(* PLC project First Steps, Beremiz Beremiz 1 *)
(* stored: creationDateTime 2016-10-24T18:09:22, modificationDateTime 2024-12-18T14:47:09 *)

PROGRAM plc_prg
  VAR
    LocalVar0 : DINT := 0;
  END_VAR
  VAR
    LocalVar1 AT %QD0.2 : DINT;
    LocalVar2 AT %ID0.2 : DINT;
  END_VAR
  VAR
    python_eval0 : python_eval;
    python_eval1 : python_eval;
  END_VAR
  VAR  (* added by the conversion: wires and edge detectors of the diagram *)
    _GT8_OUT : BOOL;
  END_VAR

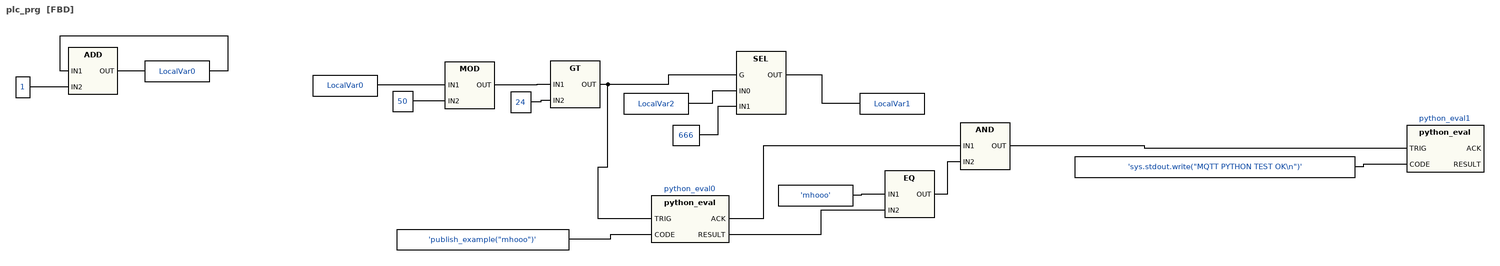
(* FBD diagram, written out as Structured Text *)
LocalVar0 := LocalVar0 + 1;
_GT8_OUT := LocalVar0 MOD 50 > 24;
LocalVar1 := SEL(_GT8_OUT, LocalVar2, 666);
python_eval0(TRIG := _GT8_OUT, CODE := 'publish_example("mhooo")');
python_eval1(TRIG := python_eval0.ACK AND 'mhooo' = python_eval0.RESULT, CODE := 'sys.stdout.write("MQTT PYTHON TEST OK\n")');
END_PROGRAM

CONFIGURATION config
  VAR_GLOBAL CONSTANT
    ResetCounterValue : INT := 17;
  END_VAR
  RESOURCE resource1 ON PLC
    TASK plc_task(INTERVAL := T#100ms, PRIORITY := 1);
    PROGRAM plc_task_instance WITH plc_task : plc_prg;
  END_RESOURCE
END_CONFIGURATION
